{attribute 'linkalways'} 
{attribute 'no_explicit_call' := 'This FB is a CLASS and must be accessed using methods or properties'}
{attribute 'enable_dynamic_creation'}
FUNCTION_BLOCK _ETcVnSvmSgdClassifierType EXTENDS EnumDatatypeBase
VAR
	localData : ETcVnSvmSgdClassifierType;
	activeData : REFERENCE TO ETcVnSvmSgdClassifierType;
	enumBaseDatatype : _DINT(localData);
END_VAR

METHOD PRIVATE AddLocalEnumeration
VAR_INPUT
	Enumeration : T_MAXSTRING;
	Value : ETcVnSvmSgdClassifierType;
END_VAR
AddEnumeration(Enumeration, Value);
END_METHOD

PROPERTY PUBLIC Address : PVOID
GET
Address := ADR(activeData);
END_GET
END_PROPERTY

METHOD PUBLIC ClearReference
VAR_INPUT
END_VAR
activeData REF= localData;
SetBaseDatatypeReference();
END_METHOD

METHOD PUBLIC Clone : I_Datatype
VAR
    pClone : POINTER TO _ETcVnSvmSgdClassifierType;
END_VAR
pClone := __NEW(_ETcVnSvmSgdClassifierType(InitialValue := Value));
Clone := pClone^;
END_METHOD

METHOD FB_init : BOOL
VAR_INPUT
	bInitRetains : BOOL; // if TRUE, the retain variables are initialized (warm start / cold start)
	bInCopyCode : BOOL;  // if TRUE, the instance afterwards gets moved into the copy code (online change)
	InitialValue : ETcVnSvmSgdClassifierType;
END_VAR
localData := InitialValue;
AddBaseDatatype(enumBaseDatatype);
ClearReference();

AddLocalEnumeration('TCVN_SSCT_SGD', ETcVnSvmSgdClassifierType.TCVN_SSCT_SGD);
AddLocalEnumeration('TCVN_SSCT_ASGD', ETcVnSvmSgdClassifierType.TCVN_SSCT_ASGD);
END_METHOD

PROPERTY PUBLIC Identifier : T_MAXSTRING
GET
Identifier := 'ETcVnSvmSgdClassifierType';
END_GET
END_PROPERTY

METHOD IsEnumeratorValueEqual : BOOL
VAR_INPUT
	Enumerator : I_KeyValueForwardEnumerator;
END_VAR
VAR
	storedValue : ETcVnSvmSgdClassifierType;
END_VAR
IF NOT Enumerator.TryGet(storedValue) THEN
	RETURN;
END_IF

IsEnumeratorValueEqual := storedValue = activeData;
END_METHOD

METHOD PUBLIC MakeReferenceTo
VAR_INPUT
	ReferenceTarget : REFERENCE TO ETcVnSvmSgdClassifierType;
END_VAR
activeData REF= ReferenceTarget;
SetBaseDatatypeReference();
END_METHOD

METHOD PROTECTED SetBaseDatatypeReference
VAR_INPUT
END_VAR
enumBaseDatatype.MakeReferenceTo(activeData);
END_METHOD

PROPERTY PUBLIC Size : UDINT
GET
Size := SIZEOF(activeData);
END_GET
END_PROPERTY

METHOD TryMakeReferenceTo : BOOL
VAR_INPUT
	Target : I_Datatype;
END_VAR
VAR
	targetAsEnum : I_EnumDatatype;
	pTargetData : POINTER TO ETcVnSvmSgdClassifierType;
END_VAR
IF NOT Target.TryResolveAsEnumDatatype(targetAsEnum) THEN
	RETURN;
END_IF

IF targetAsEnum.Identifier <> Identifier THEN
	RETURN;
END_IF

pTargetData := Target.Address;
activeData REF= pTargetData^;
SetBaseDatatypeReference();
TryMakeReferenceTo := TRUE;
END_METHOD

PROPERTY PUBLIC Value : ETcVnSvmSgdClassifierType
GET
Value := activeData;
END_GET
SET
activeData := Value;
END_SET
END_PROPERTY

END_FUNCTION_BLOCK

(* stored: Version 1.1.0.1, ProductVersion 3.1.4024.13
   POU _ETcVnSvmSgdClassifierType: Id {c5518345-f3e1-0ded-0cb1-e777a8c02e79}, SpecialFunc None
   Folder Core: Id {0caba2de-8c3c-0760-0756-7405af98abda}
   Folder Protected: Id {3f09a59f-3834-05ec-3cd2-9be0a397f293}
   Folder Customize: Id {e0a59d03-a33b-0801-08e6-80f56727a59c}
   Folder Constructor: Id {291db5c4-92fa-0bf9-2d5b-7faace861b83}
   Folder Private: Id {ff5fd792-bbd9-04a5-1d4c-239bed660d2d}
   Folder Protected: Id {7466831e-2bd8-0773-02a2-06ec616a91bd}
   Method AddLocalEnumeration: Id {6bc7ab7d-e11f-0773-1ce2-d5454ee537ab}
   Property Address: Id {3869bbff-ac2e-0987-185b-d517b32ee868}
   Get Get: Id {6fd7c906-180d-0322-1a90-8af69bb786a1}
   Method ClearReference: Id {2f87c926-a2e0-05cf-296a-1ccb4c0a28ca}
   Method Clone: Id {11b1ea59-b3a1-0527-1b17-198c22c7b21f}
   Method FB_init: Id {8550c557-9e51-0161-03ff-b1ecf1a48d17}
   Property Identifier: Id {494ba0ba-5775-0b49-2faa-e1361d3d15d1}
   Get Get: Id {91eb612b-300e-04ea-0da6-afe3d2055e65}
   Method IsEnumeratorValueEqual: Id {0545ba94-bdd7-054c-1579-0818c0c4a302}
   Method MakeReferenceTo: Id {a3bda706-b471-0bee-2adc-1c26032e7f80}
   Method SetBaseDatatypeReference: Id {f175f0ac-572d-06f2-3d87-86097707fb6f}
   Property Size: Id {2363963d-8297-0ffd-301a-3dcf4da5897c}
   Get Get: Id {742b6036-aae0-0fa9-0cca-4321c8ee4267}
   Method TryMakeReferenceTo: Id {2e8720c5-814e-0086-1717-bf54aae5cf44}
   Property Value: Id {a0026781-22e9-04b8-09ad-f55dc019b4b5}
   Get Get: Id {6f36f250-b65a-0702-2577-f651f4b227bd}
   Set Set: Id {dbe620df-3a2e-05a7-1bbd-00c9f3fd927c} *)
